Staubli VAL3: getActiveJob.pgx

public program getActiveJob(num handle_, string& value_[], bool& result_[])
begin
  // read current active job
  //
  nCommand[handle_]=coGF
  call sendCommand(handle_,"gf",result_)
  if result_
    call readSocket(handle_,value_,result_)
  else
    value_=""
  endIf
end
